(* IEC 61131-3 sources: AXOpen/src/components.festo.drives/app/src/Documentation, 4 files *)

(* ---- Component_1.st ---- *)
USING AXOpen.Components.Abstractions.Drives;
USING AXOpen.Core;

NAMESPACE AXOpen.Components.Festo.Drives
    {S7.extern=ReadWrite}
    CLASS Component_1 EXTENDS AXOpen.Core.AxoObject
        //<ComponentDeclaration>
        VAR PUBLIC
            AxoCmmtAs : AXOpen.Components.Festo.Drives.AxoCmmtAs;
        END_VAR
        //</ComponentDeclaration>

        //<InitializationArgumentsDeclaration>
        VAR PUBLIC
            manualControl   :   BOOL;
            Enable          :   BOOL;                       //  As long as ‘Enable’ is true, power is being enabled.
            EnablePositive  :   BOOL;                       //  As long as ‘Enable’ is true, this permits motion in positive direction
            EnableNegative  :   BOOL;                       //  As long as ‘Enable’ is true, this permits motion in negative direction
        END_VAR
        //</InitializationArgumentsDeclaration>

        METHOD PUBLIC Run
            VAR_INPUT
                parent : IAxoContext;
            END_VAR
            // RETURN;

            THIS.InitializeWithContext(parent);

            IF(manualControl) THEN
                AxoCmmtAs.ActivateManualControl();
            END_IF;

            //<Initialization>
            AxoCmmtAs.Run(parent            :=  THIS,
                            hwID                  :=    HwIdentifiers#cmmtas_HwID,
                            hwIdTelegram111       :=    HwIdentifiers#cmmtas_SiemensTelegram111_PZD_12_12_HwID,
                            hwIdTelegram750       :=    HwIdentifiers#cmmtas_SiemensTelegram750_PZD_4_1_HwID,
                            MAP_HW_ID             :=    HwIdentifiers#cmmtas_cmmtas_DoServo_Module_Access_Point_HwID,
                            Enable                :=    Enable,
                            EnablePositive        :=    EnablePositive,
                            EnableNegative        :=    EnableNegative);
            //</Initialization>
            THIS.UseInSequencer();

        END_METHOD

        //<Usage>
        VAR PUBLIC
            Sequencer : AxoSequencer;
            Steps : ARRAY[0..30] OF AXOpen.Core.AxoStep;
        END_VAR

        VAR PRIVATE
            _Valid : BOOL;
            _BoolValue  : BOOL;
            _DintValue  : DINT;
            _RealValue  : REAL;
            _i          : INT;
            _TaskState  :   IAxoTaskState;
        END_VAR
        METHOD PRIVATE UseInSequencer

            Sequencer.Initialize(THIS);
            Sequencer.Open();
            Sequencer.SequenceMode := eAxoSequenceMode#RunOnce;

            _i := 0;
            IF(Steps[_i].Execute(Sequencer, 'Restore')) THEN
                manualControl := FALSE;
                Enable := FALSE;
                EnablePositive := FALSE;
                EnableNegative := FALSE;
                AxoCmmtAs.Restore();
                Sequencer.MoveNext();
            END_IF;

            _i := _i + 1;
            IF(Steps[_i].Execute(Sequencer, 'Reset drive')) THEN
                IF(AxoCmmtAs.AxoReset().IsDone()) THEN
                    Sequencer.MoveNext();
                END_IF;
            END_IF;

            _i := _i + 1;
            IF(Steps[_i].Execute(Sequencer, 'Enable drive')) THEN
                Enable := TRUE;
                EnablePositive := TRUE;
                EnableNegative := TRUE;
                IF(AxoCmmtAs.AxoPower_Status) THEN
                    Sequencer.MoveNext();
                END_IF;
            END_IF;

            _i := _i + 1;
            IF(Steps[_i].Execute(Sequencer, 'Drive homming')) THEN
                IF(AxoCmmtAs.AxoHome(  Position        :=  LREAL#0.005,
                                            HommingMode     :=  INT#-17,
                                            Velocity        :=  LREAL#0.01,
                                            Acceleration    :=  LREAL#1.0,
                                            Deceleration    :=  LREAL#1.0
                                            ).IsDone()) THEN
                    Sequencer.MoveNext();
                    AxoCmmtAs.Restore();
                END_IF;
            END_IF;

            _i := _i + 1;
            IF(Steps[_i].Execute(Sequencer, 'Check position')) THEN
                IF(AxoCmmtAs.ActualPosition >=0.0049 AND  AxoCmmtAs.ActualPosition <=0.0051) THEN
                    Sequencer.MoveNext();
                END_IF;
            END_IF;

            _i := _i + 1;
            IF(Steps[_i].Execute(Sequencer, 'Set position')) THEN
                IF(AxoCmmtAs.AxoSetPosition(Position :=  LREAL#0.0).IsDone()) THEN
                    Sequencer.MoveNext();
                    AxoCmmtAs.Restore();
                END_IF;
            END_IF;

            _i := _i + 1;
            IF(Steps[_i].Execute(Sequencer, 'Check position')) THEN
                IF(AxoCmmtAs.ActualPosition >=-0.0001 AND  AxoCmmtAs.ActualPosition <=0.0001) THEN
                    Sequencer.MoveNext();
                END_IF;
            END_IF;

            _i := _i + 1;
            IF(Steps[_i].Execute(Sequencer, 'Move absolute')) THEN
                IF(AxoCmmtAs.AxoMoveAbsolute(  Position        :=  LREAL#0.005,
                                                    Velocity        :=  LREAL#0.3,
                                                    Acceleration    :=  LREAL#1.0,
                                                    Deceleration    :=  LREAL#1.0,
                                                    Jerk            :=  LREAL#500.0
                                                    ).IsDone()) THEN
                    Sequencer.MoveNext();
                    AxoCmmtAs.Restore();
                END_IF;
            END_IF;

            _i := _i + 1;
            IF(Steps[_i].Execute(Sequencer, 'Check position')) THEN
                IF(AxoCmmtAs.ActualPosition >=0.0049 AND  AxoCmmtAs.ActualPosition <=0.0051) THEN
                    Sequencer.MoveNext();
                END_IF;
            END_IF;

            _i := _i + 1;
            IF(Steps[_i].Execute(Sequencer, 'Move additive')) THEN
                AxoCmmtAs.AxoMoveAbsolute(  Position           :=  LREAL#0.010,
                                                    Velocity        :=  LREAL#0.3,
                                                    Acceleration    :=  LREAL#1.0,
                                                    Deceleration    :=  LREAL#1.0,
                                                    Jerk            :=  LREAL#500.0
                                                    );
                IF AxoCmmtAs.ActualPosition > 0.006 THEN
                    AxoCmmtAs.AxoMoveAdditive(  Distance        :=  LREAL#0.005,
                                                        Velocity        :=  LREAL#0.1,
                                                        Acceleration    :=  LREAL#1.0,
                                                        Deceleration    :=  LREAL#1.0,
                                                        Jerk            :=  LREAL#500.0
                                                        );
                END_IF;
                IF(AxoCmmtAs.AxoMoveAdditive_Task.IsDone()) THEN
                        Sequencer.MoveNext();
                        AxoCmmtAs.Restore();
                END_IF;
            END_IF;

            _i := _i + 1;
            IF(Steps[_i].Execute(Sequencer, 'Check position')) THEN
                IF(AxoCmmtAs.ActualPosition >=0.0149 AND  AxoCmmtAs.ActualPosition <=0.0151) THEN
                    Sequencer.MoveNext();
                END_IF;
            END_IF;

            _i := _i + 1;
            IF(Steps[_i].Execute(Sequencer, 'Move relative')) THEN
                IF(AxoCmmtAs.AxoMoveRelative(  Distance        :=  LREAL#-0.0050,
                                                    Velocity        :=  LREAL#0.10,
                                                    Acceleration    :=  LREAL#1.0,
                                                    Deceleration    :=  LREAL#1.0,
                                                    Jerk            :=  LREAL#500.0
                                                    ).IsDone()) THEN
                    Sequencer.MoveNext();
                    AxoCmmtAs.Restore();
                END_IF;
            END_IF;

            _i := _i + 1;
            IF(Steps[_i].Execute(Sequencer, 'Check position')) THEN
                IF(AxoCmmtAs.ActualPosition >=0.0099 AND  AxoCmmtAs.ActualPosition <=0.0101) THEN
                    Sequencer.MoveNext();
                END_IF;
            END_IF;

            _i := _i + 1;
            IF(Steps[_i].Execute(Sequencer, 'Read digital input')) THEN
                AxoCmmtAs.AxoReadDigitalInput(Enable := TRUE, InputNumber := 2 , Valid=> _Valid, Value => _BoolValue);
                IF(_Valid AND _BoolValue) THEN
                    Sequencer.MoveNext();
                    AxoCmmtAs.AxoReadDigitalInput(Enable :=FALSE);
                    AxoCmmtAs.Restore();
                END_IF;
            END_IF;

            _i := _i + 1;
            IF(Steps[_i].Execute(Sequencer, 'Move velocity')) THEN
                AxoCmmtAs.AxoMoveVelocity(  Velocity        :=  LREAL#0.01,
                                                    Acceleration    :=  LREAL#1.0,
                                                    Deceleration    :=  LREAL#1.0,
                                                    Jerk            :=  LREAL#500.0,
                                                    Direction       :=  eAxoDriveDirection#NegativeDirection,
                                                    InVelocity      => _BoolValue);
                IF(_BoolValue) THEN
                    Sequencer.MoveNext();
                    AxoCmmtAs.Restore();
                END_IF;
            END_IF;

            _i := _i + 1;
            IF(Steps[_i].Execute(Sequencer, 'Halt')) THEN
                IF(AxoCmmtAs.AxoHalt(   Deceleration    :=  LREAL#1.0,
                                        Jerk            :=  LREAL#500.0
                                        ).IsDone()) THEN
                    Sequencer.MoveNext();
                    AxoCmmtAs.Restore();
                    RETURN;
                END_IF;
            END_IF;

            _i := _i + 1;
            IF(Steps[_i].Execute(Sequencer, 'Move velocity')) THEN
                AxoCmmtAs.AxoMoveVelocity(  Velocity        :=  LREAL#0.01,
                                                    Acceleration    :=  LREAL#1.0,
                                                    Deceleration    :=  LREAL#1.0,
                                                    Jerk            :=  LREAL#500.0,
                                                    Direction       :=  eAxoDriveDirection#PositiveDirection,
                                                    InVelocity      => _BoolValue);
                IF(_BoolValue) THEN
                    Sequencer.MoveNext();
                    AxoCmmtAs.Restore();
                END_IF;
            END_IF;

            _i := _i + 1;
            IF(Steps[_i].Execute(Sequencer, 'Read digital input')) THEN
                AxoCmmtAs.AxoReadDigitalInput(Enable := TRUE, InputNumber := 2 , Valid=> _Valid, Value => _BoolValue);
                IF(_Valid AND _BoolValue) THEN
                    Sequencer.MoveNext();
                    AxoCmmtAs.AxoReadDigitalInput(Enable :=FALSE);
                    AxoCmmtAs.Restore();
                END_IF;
            END_IF;

            _i := _i + 1;
            IF(Steps[_i].Execute(Sequencer, 'Disable drive')) THEN
                Enable := FALSE;
                EnablePositive := TRUE;
                EnableNegative := TRUE;
                IF(NOT AxoCmmtAs.AxoPower_Status) THEN
                    Sequencer.MoveNext();
                END_IF;
            END_IF;

            _i := _i + 1;
            IF(Steps[_i].Execute(Sequencer, 'Reset drive')) THEN
                AxoCmmtAs.AxoReset();
                Sequencer.MoveNext();
            END_IF;

            _i := _i + 1;
            IF(Steps[_i].Execute(Sequencer, 'Enable drive')) THEN
                Enable := TRUE;
                EnablePositive := TRUE;
                EnableNegative := TRUE;
                IF(AxoCmmtAs.AxoPower_Status) THEN
                    Sequencer.MoveNext();
                END_IF;
            END_IF;

            _i := _i + 1;
            IF(Steps[_i].Execute(Sequencer, 'Jog')) THEN
                manualControl := TRUE;
                AxoCmmtAs.AxoJogPositive.RemoteSwitchOn := AxoCmmtAs.ActualPosition <= 0.02;
                AxoCmmtAs.AxoJog_Velocity      :=  LREAL#0.01;
                AxoCmmtAs.AxoJog_Acceleration  :=  LREAL#1.0;
                AxoCmmtAs.AxoJog_Deceleration  :=  LREAL#1.0;
                AxoCmmtAs.AxoJog_Jerk          :=  LREAL#100.0;
                AxoCmmtAs.AxoJog_Direction     :=  AXOpen.Components.Abstractions.Drives.eAxoDriveDirection#PositiveDirection;

                IF(AxoCmmtAs.ActualPosition > 0.02) THEN
                    AxoCmmtAs.AxoJogPositive.RemoteSwitchOn := FALSE;
                END_IF;
                IF(AxoCmmtAs.ActualPosition > 0.02 AND AxoCmmtAs.AxoHalt_Done) THEN
                    Sequencer.MoveNext();
                    manualControl := FALSE;
                END_IF;
            END_IF;

            _i := _i + 1;
            IF(Steps[_i].Execute(Sequencer, 'Torque control')) THEN
                AxoCmmtAs.AxoTorqueControl(     Torque          := LREAL#0.6 ,
                                                TorqueRamp      := LREAL#1.0 ,
                                                PositionLimit   :=  LREAL#0.100,
                                                Velocity        :=  LREAL#1.0,
                                                Acceleration    :=  LREAL#1.0,
                                                Deceleration    :=  LREAL#1.0,
                                                Jerk            :=  LREAL#500.0,
                                                Direction       :=  eAxoDriveDirection#PositiveDirection,
                                                InTorque      => _BoolValue);
                IF(_BoolValue) THEN
                    Sequencer.MoveNext();
                    AxoCmmtAs.Restore();
                END_IF;
            END_IF;

            _i := _i + 1;
            IF(Steps[_i].Execute(Sequencer, 'Check position')) THEN
                IF(AxoCmmtAs.ActualPosition >=0.0021) THEN
                    Sequencer.MoveNext();
                END_IF;
            END_IF;

            _i := _i + 1;
            IF(Steps[_i].Execute(Sequencer, 'Stop')) THEN
                AxoCmmtAs.AxoStop(  Deceleration    :=  LREAL#1.0,
                                            Jerk            :=  LREAL#500.0,
                                            Done      => _BoolValue);
                IF(_BoolValue) THEN
                    Sequencer.MoveNext();
                END_IF;
            END_IF;

            _i := _i + 1;
            IF(Steps[_i].Execute(Sequencer, 'Release stop')) THEN
                AxoCmmtAs.AxoStop_Task.Restore();
                IF(AxoCmmtAs.AxoStop_Task.IsReady()) THEN
                    Sequencer.MoveNext();
                END_IF;
            END_IF;

            _i := _i + 1;
            IF(Steps[_i].Execute(Sequencer, 'Move absolute')) THEN
                IF(AxoCmmtAs.AxoMoveAbsolute(  Position        :=  LREAL#0.0,
                                                    Velocity        :=  LREAL#0.5,
                                                    Acceleration    :=  LREAL#1.0,
                                                    Deceleration    :=  LREAL#1.0,
                                                    Jerk            :=  LREAL#500.0
                                                    ).IsDone()) THEN
                    Sequencer.MoveNext();
                    AxoCmmtAs.Restore();
                END_IF;
            END_IF;

            _i := _i + 1;
            IF(Steps[_i].Execute(Sequencer, 'Disable drive')) THEN
                Enable := FALSE;
                EnablePositive := FALSE;
                EnableNegative := FALSE;
                IF(NOT AxoCmmtAs.AxoPower_Status) THEN
                    Sequencer.MoveNext();
                END_IF;
            END_IF;

            _i := _i + 1;
            IF(Steps[_i].Execute(Sequencer, 'Reset drive')) THEN
                IF(AxoCmmtAs.AxoReset().IsDone()) THEN
                    Sequencer.MoveNext();
                END_IF;
            END_IF;

            _i := _i + 1;
            IF(Steps[_i].Execute(Sequencer, 'Restore')) THEN
                AxoCmmtAs.Restore();
                Sequencer.CompleteSequence();
            END_IF;
        END_METHOD
        // </Usage>
    END_CLASS
END_NAMESPACE

(* ---- Component_2.st ---- *)
USING AXOpen.Components.Abstractions.Drives;
USING AXOpen.Core;

NAMESPACE AXOpen.Components.Festo.Drives
    {S7.extern=ReadWrite}
    CLASS Component_2 EXTENDS AXOpen.Core.AxoObject
        //<ComponentDeclaration>
        VAR PUBLIC
            AxoCmmtAs : AXOpen.Components.Festo.Drives.AxoCmmtAs;
        END_VAR
        //</ComponentDeclaration>

        //<InitializationArgumentsDeclaration>
        VAR PUBLIC
            manualControl   :   BOOL;
            Enable          :   BOOL;                       //  As long as ‘Enable’ is true, power is being enabled.
            EnablePositive  :   BOOL;                       //  As long as ‘Enable’ is true, this permits motion in positive direction
            EnableNegative  :   BOOL;                       //  As long as ‘Enable’ is true, this permits motion in negative direction
        END_VAR
        //</InitializationArgumentsDeclaration>

        METHOD PUBLIC Run
            VAR_INPUT
                parent : IAxoContext;
            END_VAR

            THIS.InitializeWithContext(parent);

            IF(manualControl) THEN
                AxoCmmtAs.ActivateManualControl();
            END_IF;

            //<Initialization>
            AxoCmmtAs.Run(parent            :=  THIS,
                            hwID                  :=    HwIdentifiers#cmmtas_HwID,
                            hwIdTelegram111       :=    HwIdentifiers#cmmtas_SiemensTelegram111_PZD_12_12_HwID,
                            hwIdTelegram750       :=    HwIdentifiers#cmmtas_SiemensTelegram750_PZD_4_1_HwID,
                            MAP_HW_ID             :=    HwIdentifiers#cmmtas_cmmtas_DoServo_Module_Access_Point_HwID,
                            Enable                :=    Enable,
                            EnablePositive        :=    EnablePositive,
                            EnableNegative        :=    EnableNegative);
            //</Initialization>
            THIS.UseInSequencer();

        END_METHOD

        //<Usage>
        VAR PUBLIC
            Sequencer : AxoSequencer;
            Steps : ARRAY[0..30] OF AXOpen.Core.AxoStep;
        END_VAR

        VAR PRIVATE
            _Valid : BOOL;
            _BoolValue  : BOOL;
            _DintValue  : DINT;
            _RealValue  : REAL;
            _i          : INT;
            _TaskState  :   IAxoTaskState;
        END_VAR
        METHOD PRIVATE UseInSequencer

            Sequencer.Initialize(THIS);
            Sequencer.Open();
            Sequencer.SequenceMode := eAxoSequenceMode#RunOnce;

            _i := 0;
            IF(Steps[_i].Execute(Sequencer, 'Restore')) THEN
                manualControl := FALSE;
                Enable := FALSE;
                EnablePositive := FALSE;
                EnableNegative := FALSE;
                AxoCmmtAs.Restore();
                Sequencer.MoveNext();
            END_IF;

            _i := _i + 1;
            IF(Steps[_i].Execute(Sequencer, 'Reset drive')) THEN
                IF(AxoCmmtAs.AxoReset().IsDone()) THEN
                    Sequencer.MoveNext();
                END_IF;
            END_IF;

            _i := _i + 1;
            IF(Steps[_i].Execute(Sequencer, 'Enable drive')) THEN
                Enable := TRUE;
                EnablePositive := TRUE;
                EnableNegative := TRUE;
                IF(AxoCmmtAs.AxoPower_Status) THEN
                    Sequencer.MoveNext();
                END_IF;
            END_IF;

            _i := _i + 1;
            IF(Steps[_i].Execute(Sequencer, 'Drive homming')) THEN
                IF(AxoCmmtAs.AxoHome(  Position        :=  LREAL#0.005,
                                            HommingMode     :=  INT#-17,
                                            Velocity        :=  LREAL#0.01,
                                            Acceleration    :=  LREAL#1.0,
                                            Deceleration    :=  LREAL#1.0
                                            ).IsDone()) THEN
                    Sequencer.MoveNext();
                END_IF;
            END_IF;

            _i := _i + 1;
            IF(Steps[_i].Execute(Sequencer, 'Check position')) THEN
                IF(AxoCmmtAs.ActualPosition >=0.0049 AND  AxoCmmtAs.ActualPosition <=0.0051) THEN
                    Sequencer.MoveNext();
                END_IF;
            END_IF;

            _i := _i + 1;
            IF(Steps[_i].Execute(Sequencer, 'Set position')) THEN
                IF(AxoCmmtAs.AxoSetPosition(Position :=  LREAL#0.0).IsDone()) THEN
                    Sequencer.MoveNext();
                END_IF;
            END_IF;

            _i := _i + 1;
            IF(Steps[_i].Execute(Sequencer, 'Check position')) THEN
                IF(AxoCmmtAs.ActualPosition >=-0.0001 AND  AxoCmmtAs.ActualPosition <=0.0001) THEN
                    Sequencer.MoveNext();
                END_IF;
            END_IF;

            _i := _i + 1;
            IF(Steps[_i].Execute(Sequencer, 'Move absolute')) THEN
                IF(AxoCmmtAs.AxoMoveAbsolute(  Position        :=  LREAL#0.005,
                                                    Velocity        :=  LREAL#0.3,
                                                    Acceleration    :=  LREAL#1.0,
                                                    Deceleration    :=  LREAL#1.0,
                                                    Jerk            :=  LREAL#500.0
                                                    ).IsDone()) THEN
                    Sequencer.MoveNext();
                    AxoCmmtAs.AxoMoveAbsolute_Task.Restore();
                    RETURN;
                END_IF;
            END_IF;

            _i := _i + 1;
            IF(Steps[_i].Execute(Sequencer, 'Check position')) THEN
                IF(AxoCmmtAs.ActualPosition >=0.0049 AND  AxoCmmtAs.ActualPosition <=0.0051) THEN
                    Sequencer.MoveNext();
                END_IF;
            END_IF;

            _i := _i + 1;
            IF(Steps[_i].Execute(Sequencer, 'Move additive')) THEN
                AxoCmmtAs.AxoMoveAbsolute(  Position           :=  LREAL#0.010,
                                                    Velocity        :=  LREAL#0.3,
                                                    Acceleration    :=  LREAL#1.0,
                                                    Deceleration    :=  LREAL#1.0,
                                                    Jerk            :=  LREAL#500.0
                                                    );
                IF AxoCmmtAs.ActualPosition > 0.006 THEN
                    AxoCmmtAs.AxoMoveAdditive(  Distance        :=  LREAL#0.005,
                                                        Velocity        :=  LREAL#0.1,
                                                        Acceleration    :=  LREAL#1.0,
                                                        Deceleration    :=  LREAL#1.0,
                                                        Jerk            :=  LREAL#500.0
                                                        );
                END_IF;
                IF(AxoCmmtAs.AxoMoveAdditive_Task.IsDone()) THEN
                        Sequencer.MoveNext();
                END_IF;
            END_IF;

            _i := _i + 1;
            IF(Steps[_i].Execute(Sequencer, 'Check position')) THEN
                IF(AxoCmmtAs.ActualPosition >=0.0149 AND  AxoCmmtAs.ActualPosition <=0.0151) THEN
                    Sequencer.MoveNext();
                END_IF;
            END_IF;

            _i := _i + 1;
            IF(Steps[_i].Execute(Sequencer, 'Move relative')) THEN
                IF(AxoCmmtAs.AxoMoveRelative(  Distance        :=  LREAL#-0.0050,
                                                    Velocity        :=  LREAL#0.10,
                                                    Acceleration    :=  LREAL#1.0,
                                                    Deceleration    :=  LREAL#1.0,
                                                    Jerk            :=  LREAL#500.0
                                                    ).IsDone()) THEN
                    Sequencer.MoveNext();
                END_IF;
            END_IF;

            _i := _i + 1;
            IF(Steps[_i].Execute(Sequencer, 'Check position')) THEN
                IF(AxoCmmtAs.ActualPosition >=0.0099 AND  AxoCmmtAs.ActualPosition <=0.0101) THEN
                    Sequencer.MoveNext();
                END_IF;
            END_IF;

            _i := _i + 1;
            IF(Steps[_i].Execute(Sequencer, 'Read digital input')) THEN
                AxoCmmtAs.AxoReadDigitalInput(Enable := TRUE, InputNumber := 2 , Valid=> _Valid, Value => _BoolValue);
                IF(_Valid AND _BoolValue) THEN
                    Sequencer.MoveNext();
                    AxoCmmtAs.AxoReadDigitalInput(Enable :=FALSE);
                END_IF;
            END_IF;

            _i := _i + 1;
            IF(Steps[_i].Execute(Sequencer, 'Move velocity')) THEN
                AxoCmmtAs.AxoMoveVelocity(  Velocity        :=  LREAL#0.01,
                                                    Acceleration    :=  LREAL#1.0,
                                                    Deceleration    :=  LREAL#1.0,
                                                    Jerk            :=  LREAL#500.0,
                                                    Direction       :=  eAxoDriveDirection#NegativeDirection,
                                                    InVelocity      => _BoolValue);
                IF(_BoolValue) THEN
                    Sequencer.MoveNext();
                    AxoCmmtAs.AxoMoveVelocity_Task.Restore();
                    RETURN;
                END_IF;
            END_IF;

            _i := _i + 1;
            IF(Steps[_i].Execute(Sequencer, 'Halt')) THEN
                IF(AxoCmmtAs.AxoHalt(  Deceleration    :=  LREAL#1.0,
                                            Jerk            :=  LREAL#500.0
                                            ).IsDone()) THEN
                    Sequencer.MoveNext();
                END_IF;
            END_IF;

            _i := _i + 1;
            IF(Steps[_i].Execute(Sequencer, 'Move velocity')) THEN
                AxoCmmtAs.AxoMoveVelocity(  Velocity        :=  LREAL#0.01,
                                                    Acceleration    :=  LREAL#1.0,
                                                    Deceleration    :=  LREAL#1.0,
                                                    Jerk            :=  LREAL#500.0,
                                                    Direction       :=  eAxoDriveDirection#PositiveDirection,
                                                    InVelocity      => _BoolValue);
                IF(_BoolValue) THEN
                    Sequencer.MoveNext();
                END_IF;
            END_IF;

            _i := _i + 1;
            IF(Steps[_i].Execute(Sequencer, 'Read digital input')) THEN
                AxoCmmtAs.AxoReadDigitalInput(Enable := TRUE, InputNumber := 2 , Valid=> _Valid, Value => _BoolValue);
                IF(_Valid AND _BoolValue) THEN
                    Sequencer.MoveNext();
                    AxoCmmtAs.AxoReadDigitalInput(Enable :=FALSE);
                END_IF;
            END_IF;

            _i := _i + 1;
            IF(Steps[_i].Execute(Sequencer, 'Disable drive')) THEN
                Enable := FALSE;
                EnablePositive := TRUE;
                EnableNegative := TRUE;
                IF(NOT AxoCmmtAs.AxoPower_Status) THEN
                    Sequencer.MoveNext();
                END_IF;
            END_IF;

            _i := _i + 1;
            IF(Steps[_i].Execute(Sequencer, 'Reset drive')) THEN
                AxoCmmtAs.AxoReset();
                Sequencer.MoveNext();
            END_IF;

            _i := _i + 1;
            IF(Steps[_i].Execute(Sequencer, 'Enable drive')) THEN
                Enable := TRUE;
                EnablePositive := TRUE;
                EnableNegative := TRUE;
                IF(AxoCmmtAs.AxoPower_Status) THEN
                    Sequencer.MoveNext();
                END_IF;
            END_IF;

            _i := _i + 1;
            IF(Steps[_i].Execute(Sequencer, 'Jog')) THEN
                manualControl := TRUE;
                AxoCmmtAs.AxoJogPositive.RemoteSwitchOn := AxoCmmtAs.ActualPosition <= 0.02;
                AxoCmmtAs.AxoJog_Velocity      :=  LREAL#0.01;
                AxoCmmtAs.AxoJog_Acceleration  :=  LREAL#1.0;
                AxoCmmtAs.AxoJog_Deceleration  :=  LREAL#1.0;
                AxoCmmtAs.AxoJog_Jerk          :=  LREAL#100.0;
                AxoCmmtAs.AxoJog_Direction     :=  AXOpen.Components.Abstractions.Drives.eAxoDriveDirection#PositiveDirection;

                IF(AxoCmmtAs.ActualPosition > 0.02) THEN
                    AxoCmmtAs.AxoJogPositive.RemoteSwitchOn := FALSE;
                END_IF;
                IF(AxoCmmtAs.ActualPosition > 0.02 AND AxoCmmtAs.AxoHalt_Done) THEN
                    Sequencer.MoveNext();
                    manualControl := FALSE;
                END_IF;
            END_IF;

            _i := _i + 1;
            IF(Steps[_i].Execute(Sequencer, 'Torque control')) THEN
                AxoCmmtAs.AxoTorqueControl(     Torque          := LREAL#0.6 ,
                                                TorqueRamp      := LREAL#1.0 ,
                                                PositionLimit   :=  LREAL#0.100,
                                                Velocity        :=  LREAL#1.0,
                                                Acceleration    :=  LREAL#1.0,
                                                Deceleration    :=  LREAL#1.0,
                                                Jerk            :=  LREAL#500.0,
                                                Direction       :=  eAxoDriveDirection#PositiveDirection,
                                                InTorque      => _BoolValue);
                IF(_BoolValue) THEN
                    Sequencer.MoveNext();
                END_IF;
            END_IF;

            _i := _i + 1;
            IF(Steps[_i].Execute(Sequencer, 'Check position')) THEN
                IF(AxoCmmtAs.ActualPosition >=0.0021) THEN
                    Sequencer.MoveNext();
                END_IF;
            END_IF;

            _i := _i + 1;
            IF(Steps[_i].Execute(Sequencer, 'Stop')) THEN
                AxoCmmtAs.AxoStop(  Deceleration    :=  LREAL#1.0,
                                            Jerk            :=  LREAL#500.0,
                                            Done      => _BoolValue);
                IF(_BoolValue) THEN
                    Sequencer.MoveNext();
                END_IF;
            END_IF;

            _i := _i + 1;
            IF(Steps[_i].Execute(Sequencer, 'Release stop')) THEN
                AxoCmmtAs.AxoStop_Task.Restore();
                IF(AxoCmmtAs.AxoStop_Task.IsReady()) THEN
                    Sequencer.MoveNext();
                END_IF;
            END_IF;

            _i := _i + 1;
            IF(Steps[_i].Execute(Sequencer, 'Move absolute')) THEN
                IF(AxoCmmtAs.AxoMoveAbsolute(  Position        :=  LREAL#0.0,
                                                    Velocity        :=  LREAL#0.5,
                                                    Acceleration    :=  LREAL#1.0,
                                                    Deceleration    :=  LREAL#1.0,
                                                    Jerk            :=  LREAL#500.0
                                                    ).IsDone()) THEN
                    Sequencer.MoveNext();
                END_IF;
            END_IF;

            _i := _i + 1;
            IF(Steps[_i].Execute(Sequencer, 'Disable drive')) THEN
                Enable := FALSE;
                EnablePositive := FALSE;
                EnableNegative := FALSE;
                IF(NOT AxoCmmtAs.AxoPower_Status) THEN
                    Sequencer.CompleteSequence();
                END_IF;
            END_IF;

            _i := _i + 1;
            IF(Steps[_i].Execute(Sequencer, 'Reset drive')) THEN
                IF(AxoCmmtAs.AxoReset().IsDone()) THEN
                    Sequencer.MoveNext();
                END_IF;
            END_IF;

            _i := _i + 1;
            IF(Steps[_i].Execute(Sequencer, 'Restore')) THEN
                AxoCmmtAs.Restore();
                Sequencer.CompleteSequence();
            END_IF;
        END_METHOD
        // </Usage>
    END_CLASS
END_NAMESPACE

(* ---- Component_3.st ---- *)
USING AXOpen.Components.Abstractions.Drives;
USING AXOpen.Core;

{S7.extern=ReadWrite}
CLASS Component_3 EXTENDS AXOpen.Core.AxoObject
    //<ComponentDeclaration>
    VAR PUBLIC
        AxoCmmtAs : AXOpen.Components.Festo.Drives.AxoCmmtAs;
    END_VAR
    //</ComponentDeclaration>

    //<InitializationArgumentsDeclaration>
    VAR PUBLIC
        PlcInputs : REF_TO PlcInputs;
        PlcOutputs : REF_TO PlcOutputs;

        run_            :   BOOL := FALSE;
        manualControl   :   BOOL;
        Enable          :   BOOL;                       //  As long as ‘Enable’ is true, power is being enabled.
        EnablePositive  :   BOOL;                       //  As long as ‘Enable’ is true, this permits motion in positive direction
        EnableNegative  :   BOOL;                       //  As long as ‘Enable’ is true, this permits motion in negative direction
    END_VAR
    //</InitializationArgumentsDeclaration>

    METHOD PUBLIC Run
        VAR_INPUT
            parent : IAxoContext;
        END_VAR

        IF NOT run_ THEN
            RETURN;
        END_IF;

        THIS.Initialize(parent);

        IF(manualControl) THEN
            AxoCmmtAs.ActivateManualControl();
        END_IF;

        //<Initialization>
        AxoCmmtAs.Run(  parent                :=  THIS,
                            refTelegram111_In     :=  REF(PlcInputs^.cmmtas_test_DO_SERVO_1_Siemens_telegram_111_PZD_12_12),
                            refTelegram750_In     :=  REF(PlcInputs^.cmmtas_test_DO_SERVO_1_Siemens_telegram_750_PZD_4_1),
                            refTelegram111_Out    :=  REF(PlcOutputs^.cmmtas_test_DO_SERVO_1_Siemens_telegram_111_PZD_12_12),
                            refTelegram750_Out    :=  REF(PlcOutputs^.cmmtas_test_DO_SERVO_1_Siemens_telegram_750_PZD_4_1),
                            MAP_HW_ID             :=  HwIdentifiers#cmmtas_test_Module_Access_Point,
                            Enable                := Enable,
                            EnablePositive        := EnablePositive,
                            EnableNegative        := EnableNegative);
        //</Initialization>
        THIS.UseInSequencer();

    END_METHOD

    //<Usage>
    VAR PUBLIC
        Sequencer : AxoSequencer;
        Steps : ARRAY[0..16] OF AXOpen.Core.AxoStep;
    END_VAR

    VAR PRIVATE
        _Valid : BOOL;
        _BoolValue  : BOOL;
        _DintValue  : DINT;
        _RealValue  : REAL;
        _i          : INT;
        _TaskState  :   IAxoTaskState;
    END_VAR
    METHOD PRIVATE UseInSequencer

        Sequencer.Initialize(THIS);
        Sequencer.Open();
        Sequencer.SequenceMode := eAxoSequenceMode#RunOnce;

        // _i := 0;
        // IF(Steps[_i].Execute(Sequencer, 'Restore')) THEN
        //     manualControl := FALSE;
        //     // IF(AxoCmmtAsPtP_.ComponentRestore().IsDone()) THEN

        //     //            IF(AxoCmmtAsPtP_.Restore_Task.Invoke().IsDone()) THEN
        //     AxoCmmtAs.Restore();
        //         Sequencer.MoveNext();
        //     // END_IF;
        // END_IF;

        // _i := _i + 1;
        // IF(Steps[_i].Execute(Sequencer, 'Reset drive')) THEN
        //     IF(AxoCmmtAs.Reset().IsDone()) THEN
        //         Sequencer.MoveNext();
        //     END_IF;
        // END_IF;

        // _i := _i + 1;
        // IF(Steps[_i].Execute(Sequencer, 'Drive homming')) THEN
        //     IF(AxoCmmtAs.Home().IsDone()) THEN
        //         Sequencer.MoveNext();
        //     END_IF;
        // END_IF;

        // _i := _i + 1;
        // IF(Steps[_i].Execute(Sequencer, 'Check position')) THEN
        //     IF(AxoCmmtAs.ActualPosition >=-0.1 AND  AxoCmmtAs.ActualPosition <=0.1) THEN
        //         Sequencer.MoveNext();
        //     END_IF;
        // END_IF;

        // _i := _i + 1;
        // IF(Steps[_i].Execute(Sequencer, 'Move absolute')) THEN
        //     IF(AxoCmmtAs.MoveAbsolute(Position := LREAL#5.0 , Velocity := LREAL#10.0).IsDone()) THEN
        //         Sequencer.MoveNext();
        //         AxoCmmtAs.MoveAbsolute_Task.Restore();
        //         RETURN;
        //     END_IF;
        // END_IF;

        // _i := _i + 1;
        // IF(Steps[_i].Execute(Sequencer, 'Check position')) THEN
        //     IF(AxoCmmtAs.ActualPosition >=4.9 AND  AxoCmmtAs.ActualPosition <=5.1) THEN
        //         Sequencer.MoveNext();
        //     END_IF;
        // END_IF;

        // _i := _i + 1;
        // IF(Steps[_i].Execute(Sequencer, 'Move relative')) THEN
        //     IF(AxoCmmtAs.MoveRelative(Distance := LREAL#5.0 , Velocity := LREAL#10.0).IsDone()) THEN
        //         Sequencer.MoveNext();
        //     END_IF;
        // END_IF;

        // _i := _i + 1;
        // IF(Steps[_i].Execute(Sequencer, 'Check position')) THEN
        //     IF(AxoCmmtAs.ActualPosition >=9.9 AND  AxoCmmtAs.ActualPosition <=10.1) THEN
        //         Sequencer.MoveNext();
        //     END_IF;
        // END_IF;

        // _i := _i + 1;
        // IF(Steps[_i].Execute(Sequencer, 'Jog positive')) THEN
        //     manualControl := TRUE;
        //     AxoCmmtAs.JogPositive_Task.RemoteSwitchOn := TRUE;

        //     IF(AxoCmmtAs.ActualPosition > 21.0) THEN
        //         Sequencer.MoveNext();
        //         AxoCmmtAs.JogPositive_Task.RemoteSwitchOn := FALSE;
        //         manualControl := FALSE;
        //     END_IF;
        // END_IF;

        // _i := _i + 1;
        // IF(Steps[_i].Execute(Sequencer, 'Jog negative')) THEN
        //     manualControl := TRUE;
        //     AxoCmmtAs.JogNegative_Task.RemoteSwitchOn := TRUE;

        //     IF(AxoCmmtAs.ActualPosition < 20.0) THEN
        //         Sequencer.MoveNext();
        //         AxoCmmtAs.JogNegative_Task.RemoteSwitchOn := FALSE;
        //         manualControl := FALSE;
        //     END_IF;
        // END_IF;

        // _i := _i + 1;
        // IF(Steps[_i].Execute(Sequencer, 'Stop')) THEN
        //     IF (AxoCmmtAs.Stop().IsDone()) THEN
        //         Sequencer.MoveNext();
        //     END_IF;
        // END_IF;

        // _i := _i + 1;
        // IF(Steps[_i].Execute(Sequencer, 'Travel to fixed stop')) THEN
        //     _TaskState := AxoCmmtAs.TravelToFixStop(Position := LREAL#100.0 , Velocity := LREAL#5.0 , Torque := LREAL#0.5);
        //     Steps[_i].ThrowWhen(_TaskState.HasError());
        //     IF _TaskState.IsDone() OR _TaskState.HasError() THEN
        //         Sequencer.MoveNext();
        //     END_IF;
        // END_IF;

        // _i := _i + 1;
        // IF(Steps[_i].Execute(Sequencer, 'Reset drive')) THEN
        //     IF(AxoCmmtAs.Reset().IsDone()) THEN
        //         Sequencer.MoveNext();
        //     END_IF;
        // END_IF;

        // _i := _i + 1;
        // IF(Steps[_i].Execute(Sequencer, 'Move absolute')) THEN
        //     IF(AxoCmmtAs.MoveAbsolute(Position := LREAL#0.0 , Velocity := LREAL#20.0).IsDone()) THEN
        //         Sequencer.MoveNext();
        //     END_IF;
        // END_IF;

        // _i := _i + 1;
        // IF(Steps[_i].Execute(Sequencer, 'Drive homming')) THEN
        //     IF(AxoCmmtAs.Home().IsDone()) THEN
        //         Sequencer.MoveNext();
        //     END_IF;
        // END_IF;

        // _i := _i + 1;
        // IF(Steps[_i].Execute(Sequencer, 'Restore')) THEN
        //     manualControl := FALSE;
        //     IF(AxoCmmtAs.Restore_Task.Invoke().IsDone()) THEN
        //         Sequencer.CompleteSequence();
        //     END_IF;
        // END_IF;
    END_METHOD
    // </Usage>
END_CLASS

(* ---- DocumentationContext.st ---- *)
NAMESPACE AXOpen.Components.Festo.Drives
    {S7.extern=ReadWrite}
    CLASS DocumentationContext EXTENDS AXOpen.Core.AxoContext
        VAR PUBLIC
            componentOne    : Component_1;
            componentTwo    : Component_2;
        END_VAR

        METHOD PROTECTED OVERRIDE Main
            componentOne.Run(THIS);
            // componentTwo.Run(THIS);
        END_METHOD
    END_CLASS
END_NAMESPACE
